{attribute 'linkalways'} 
{attribute 'no_explicit_call' := 'This FB is a CLASS and must be accessed using methods or properties'}
{attribute 'enable_dynamic_creation'}
FUNCTION_BLOCK ABSTRACT EnumDatatypeBase EXTENDS UserDefinedDatatypeBase IMPLEMENTS I_EnumDatatype
VAR
	_baseDatatype : I_Datatype;
	enumerations : Dictionary;
END_VAR

METHOD PROTECTED AddBaseDatatype
VAR_INPUT
	BaseType : I_Datatype;
END_VAR
_baseDatatype := BaseType;
END_METHOD

METHOD PROTECTED AddEnumeration
VAR_INPUT
	Enumeration : T_MAXSTRING;
	Value : ANY;
END_VAR
enumerations.AddOrUpdate(Enumeration, Value);
END_METHOD

PROPERTY PUBLIC BaseDatatype : I_Datatype
GET
BaseDatatype := _baseDatatype;
END_GET
END_PROPERTY

METHOD PRIVATE CreateEnumError : I_Error
VAR_INPUT
	Enum : T_MAXSTRING;
END_VAR
VAR
	pError : POINTER TO UnknownEnumerationError;
END_VAR
pError := __NEW(UnknownEnumerationError(EnumString := Enum));
CreateEnumError := pError^;
END_METHOD

METHOD ABSTRACT IsEnumeratorValueEqual : BOOL
VAR_INPUT
	Enumerator : I_KeyValueForwardEnumerator;
END_VAR
END_METHOD

PROPERTY PUBLIC Name : T_MAXSTRING
GET
Name := 'ENUM';
END_GET
END_PROPERTY

METHOD PROTECTED OnSerializeTypeWith
VAR_INPUT
	Serializer : I_Serializer;
END_VAR
SUPER^.OnSerializeTypeWith(Serializer);
SerializeEnums(Serializer);
SerializeBaseType(Serializer);
END_METHOD

METHOD PRIVATE SerializeBaseType
VAR_INPUT
	Serializer : I_Serializer;
END_VAR
IF _baseDatatype = 0 THEN
	RETURN;
END_IF

Serializer.AddKey('baseType');
_baseDatatype.SerializeTypeWith(Serializer);
END_METHOD

METHOD PRIVATE SerializeEnums
VAR_INPUT
	Serializer : I_Serializer;
END_VAR
VAR
	enumerator : I_KeyValueForwardEnumerator;
END_VAR
Serializer.AddKey('enumerations');
Serializer.StartArray();

enumerator := enumerations.GetKeyValueEnumerator();

WHILE enumerator.MoveNext() DO
	Serializer.AddString(enumerator.Key);
END_WHILE

enumerator.Dispose();

Serializer.EndArray();
END_METHOD

METHOD PUBLIC SerializeWith
VAR_INPUT
	Serializer : I_Serializer;
END_VAR
VAR
	returnKey : T_MAXSTRING;
	enumerator : I_KeyValueForwardEnumerator;
END_VAR
enumerator := enumerations.GetKeyValueEnumerator();
returnKey := 'UNDEFINED';

WHILE (enumerator.MoveNext()) DO
	
	IF IsEnumeratorValueEqual(enumerator) THEN
		returnKey := enumerator.key;
		EXIT;
	END_IF

END_WHILE

Serializer.AddString(returnKey);
enumerator.Dispose();
END_METHOD

METHOD TryDeserializeFrom : BOOL
VAR_INPUT
	Deserializer : I_Deserializer;
	Feedback : I_DeserializerFeedback;
END_VAR
VAR
	key : T_MAXSTRING;
	error : I_Error;
END_VAR
IF NOT Deserializer.TryGetString(key, Feedback) THEN
	RETURN;
END_IF

IF NOT enumerations.TryGetValueTo(key, Address, Size) THEN
	error := CreateEnumError(key);
	Feedback.LogError(error);
	RETURN;
END_IF
END_METHOD

METHOD PUBLIC TryResolveAsEnumDatatype : BOOL
VAR_INPUT
	Destination : REFERENCE TO I_EnumDatatype;
END_VAR
Destination := THIS^;
TryResolveAsEnumDatatype := TRUE;
END_METHOD

END_FUNCTION_BLOCK

(* stored: Version 1.1.0.1, ProductVersion 3.1.4024.12
   POU EnumDatatypeBase: Id {fdfb72f6-54ae-016d-3ae9-df54d942308f}, SpecialFunc None
   Folder Private: Id {4ac5f28a-3d92-023a-34f1-677805bad0a9}
   Folder Protected: Id {3234e302-c3fa-0a1a-1772-92d772ea6b60}
   Method AddBaseDatatype: Id {c7c1f175-08c2-0719-1f79-f8b38ca0fd55}
   Method AddEnumeration: Id {8c2cee91-baff-0cdb-0548-32a2aa6bb6b1}
   Property BaseDatatype: Id {49354021-666b-00ef-1bb6-f1a08a604711}
   Get Get: Id {7868e332-e99f-0b71-0e99-f9feb1ce23de}
   Method CreateEnumError: Id {150c80e1-67f6-0cc5-2e1e-352746685f08}
   Method IsEnumeratorValueEqual: Id {6bd6d552-765d-0592-243d-04f5783e0d69}
   Property Name: Id {21745b08-4305-0c91-28a0-7d4bdc0f51be}
   Get Get: Id {d07c6a61-fa0a-0b92-2d64-72598b395452}
   Method OnSerializeTypeWith: Id {547cf7ae-ef21-07e4-109a-fccfaf9adaea}
   Method SerializeBaseType: Id {3dbddad6-478a-000a-3783-0c654560bce3}
   Method SerializeEnums: Id {1993820e-9082-08dd-27af-84894365a6c3}
   Method SerializeWith: Id {29525bb3-f2aa-090b-29a3-26eb75da1713}
   Method TryDeserializeFrom: Id {62902a79-a65d-029d-38d5-858c7f60c88f}
   Method TryResolveAsEnumDatatype: Id {257f8d88-70ef-0584-3d43-12a10891fa60} *)
